ADAPTER AStatusLight
  (* Standard: 61499-1 *)
  (* Version 0.0, 2008-04-22, GE, 4DIAC-Consortium *)
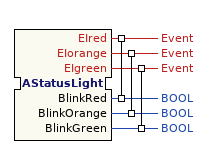
  EVENT_OUTPUT
    EIred WITH BlinkRed;
    EIorange WITH BlinkOrange;
    EIgreen WITH BlinkGreen;
  END_EVENT
  VAR_OUTPUT
    BlinkRed : BOOL;
    BlinkOrange : BOOL;
    BlinkGreen : BOOL;
  END_VAR
  SERVICE SOCKET/PLUG
    SEQUENCE request_confirm
      SOCKET.REQ(REQD) -> PLUG.REQ(REQD);
      PLUG.CNF(CNFD) -> SOCKET.CNF(CNFD);
    END_SEQUENCE
    SEQUENCE indication_response
      PLUG.IND(INDD) -> SOCKET.IND(INDD);
      SOCKET.RSP(RSPD) -> PLUG.RSP(RSPD);
    END_SEQUENCE
  END_SERVICE
END_ADAPTER
